TEXTLIST txt_opMode
  0 = 'waiting_for_calibration'
  1 = 're_init'
  2 = 'waiting'
  3 = 'moving'
  4 = 'doors_opening'
  5 = 'waiting_doors_open'
  6 = 'doors_closing'
  7 = 'PRIO waiting'
  8 = 'PRIO doors_closing'
  9 = 'PRIO moving'
  10 = 'PRIO doors_opening'
   = ''
END_TEXTLIST

(* stored: Version 1.1.0.1, ProductVersion 3.1.4024.6
   TextList txt_opMode: Id {1637e2ef-5b46-4b0b-9ee6-e32d7f5b28c3} *)
